FUNCTION_BLOCK Motor_Inversor_Automatico_Unico_HMI (* Service Interface Function Block Type *)
  (* Standard: 61499-2 *)
  (* Version 0.0, 1/22/2026, Schneider Electric, template *)
  PACKAGE Hidryco.HidrycoLib;
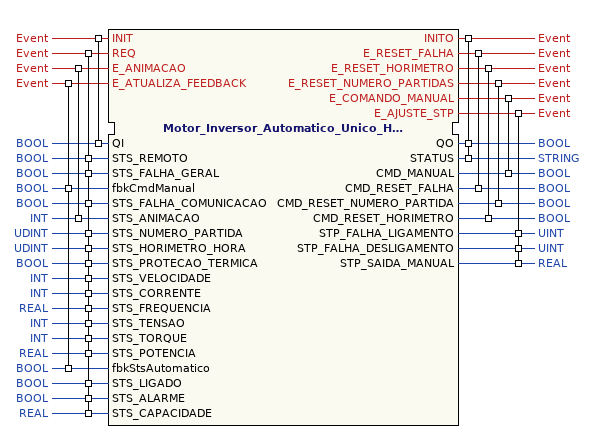
  EVENT_INPUT
    INIT WITH QI;
    REQ WITH STS_REMOTO, STS_FALHA_GERAL, STS_NUMERO_PARTIDA, STS_HORIMETRO_HORA, STS_FALHA_COMUNICACAO, STS_VELOCIDADE, STS_CORRENTE, STS_FREQUENCIA, STS_TENSAO, STS_TORQUE, STS_POTENCIA, STS_PROTECAO_TERMICA, STS_LIGADO, STS_ALARME, STS_CAPACIDADE;
    E_ANIMACAO WITH STS_ANIMACAO;
    E_ATUALIZA_FEEDBACK WITH fbkCmdManual, fbkStsAutomatico;
  END_EVENT
  EVENT_OUTPUT
    INITO WITH QO, STATUS;
    E_RESET_FALHA WITH CMD_RESET_FALHA;
    E_RESET_HORIMETRO WITH CMD_RESET_HORIMETRO;
    E_RESET_NUMERO_PARTIDAS WITH CMD_RESET_NUMERO_PARTIDA;
    E_COMANDO_MANUAL WITH CMD_MANUAL;
    E_AJUSTE_STP WITH STP_FALHA_LIGAMENTO, STP_FALHA_DESLIGAMENTO, STP_SAIDA_MANUAL;
  END_EVENT
  VAR_INPUT
    QI : BOOL;
    STS_REMOTO : BOOL;
    STS_FALHA_GERAL : BOOL;
    fbkCmdManual : BOOL;
    STS_FALHA_COMUNICACAO : BOOL;
    STS_ANIMACAO : INT;
    STS_NUMERO_PARTIDA : UDINT;
    STS_HORIMETRO_HORA : UDINT;
    STS_PROTECAO_TERMICA : BOOL;
    STS_VELOCIDADE : INT;
    STS_CORRENTE : INT;
    STS_FREQUENCIA : REAL;
    STS_TENSAO : INT;
    STS_TORQUE : INT;
    STS_POTENCIA : REAL;
    fbkStsAutomatico : BOOL;
    STS_LIGADO : BOOL;
    STS_ALARME : BOOL;
    STS_CAPACIDADE : REAL;
  END_VAR
  VAR_OUTPUT
    QO : BOOL; (* Event Output Qualifier *)
    STATUS : STRING; (* Service Status *)
    CMD_MANUAL : BOOL;
    CMD_RESET_FALHA : BOOL;
    CMD_RESET_NUMERO_PARTIDA : BOOL;
    CMD_RESET_HORIMETRO : BOOL;
    STP_FALHA_LIGAMENTO : UINT;
    STP_FALHA_DESLIGAMENTO : UINT;
    STP_SAIDA_MANUAL : REAL;
  END_VAR
  SERVICE /
    SEQUENCE 
    END_SEQUENCE
  END_SERVICE
END_FUNCTION_BLOCK
